FUNCTION_BLOCK EdgeDetect_VIEW
  (* Version 1.0, 2005-11-13, Goran Cengic, Chalmers *)
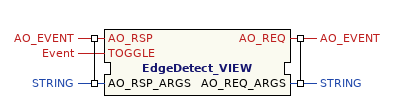
  EVENT_INPUT
    AO_RSP : AO_EVENT WITH AO_RSP_ARGS;
    TOGGLE;
  END_EVENT
  EVENT_OUTPUT
    AO_REQ : AO_EVENT WITH AO_REQ_ARGS;
  END_EVENT
  VAR_INPUT
    AO_RSP_ARGS : STRING;
  END_VAR
  VAR_OUTPUT
    AO_REQ_ARGS : STRING;
  END_VAR
  FBS
    rsp_parser : BinaryActuator_MDL_RSP_PARSE;
    req_gen : BinaryActuator_MDL_REQ_GEN;
    not : E_NOT;
  END_FBS
  EVENT_CONNECTIONS
    AO_RSP TO rsp_parser.RSP;
    rsp_parser.CURRENT_VALUE TO not.EI;
    not.EO TO req_gen.WRITE;
    req_gen.REQ TO AO_REQ;
    TOGGLE TO req_gen.CURRENT_VALUE;
  END_CONNECTIONS
  DATA_CONNECTIONS
    AO_RSP_ARGS TO rsp_parser.RSP_ARGS;
    rsp_parser.VALUE TO not.A;
    not.AN TO req_gen.VALUE;
    req_gen.REQ_ARGS TO AO_REQ_ARGS;
  END_CONNECTIONS
END_FUNCTION_BLOCK
